Yaskawa INFORM job: R1_W27-A2(90,-90)POPR-KM-OK.JBI

/JOB
//NAME R1_W27-A2(90,-90)POPR-KM-OK
///FOLDERNAME KRIS-SCIANA
//POS
///NPOS 176,176,0,6,0,0
///TOOL 0
///POSTYPE PULSE
///PULSE
C00000=47255,92390,21974,-39561,97708,85383
C00001=10855,-90008,-88389,-33686,75537,85808
C00002=-111602,-139258,-125525,-5527,77988,-30584
C00003=-111602,-139258,-125525,-5527,77988,-30584
C00004=-63451,-99780,-87259,-34493,107645,-18593
C00005=-79235,-87779,-71168,-36428,98005,-22127
C00006=-81155,-88041,-68185,-36487,95587,-22123
C00007=-83679,-90006,-68978,-36755,94086,-22676
C00008=-83320,-89737,-68871,-36718,94298,-22597
C00009=-83320,-90271,-70181,-36754,94730,-22742
C00010=-84421,-91093,-70507,-36864,94080,-22984
C00011=-84421,-90731,-69628,-36842,93792,-22887
C00012=-81728,-89912,-71997,-36675,96467,-22659
C00013=-111602,-139258,-125525,-5527,77988,-30584
C00014=-111602,-139258,-125525,-5527,77988,-30584
C00015=-131748,-141016,-124490,10531,76516,-37016
C00016=-120565,-128207,-90021,8850,60749,-34228
C00017=-114295,-127384,-89205,7232,60054,-31882
C00018=-112834,-127008,-88848,6844,59902,-31333
C00019=-110412,-126666,-88756,6184,59829,-30410
C00020=-111525,-126835,-88802,6488,59856,-30835
C00021=-111525,-128465,-91197,6450,60489,-30798
C00022=-108910,-128023,-91079,5736,60447,-29805
C00023=-108910,-126871,-89375,5761,59994,-29827
C00024=-114109,-129808,-92766,7120,60979,-31753
C00025=-125724,-137992,-104372,9805,65099,-35816
C00026=-168598,-158328,-94882,65934,65859,5142
C00027=-138330,-90233,-84655,36621,76479,52498
C00028=-128715,-49536,-61129,33505,77884,56923
C00029=-127126,-48405,-55465,33411,74823,56634
C00030=-126813,-49148,-53910,33515,73573,56377
C00031=-126089,-49251,-53971,33315,73277,56584
C00032=-126589,-49181,-53929,33454,73482,56443
C00033=-126589,-49335,-57635,33144,75338,57009
C00034=-129344,-26255,-35376,41772,85568,55954
C00035=-129533,-29426,-35674,41853,84566,55468
C00036=-129631,-31118,-36819,41874,84489,55393
C00037=-129533,-29426,-35674,41853,84566,55468
C00038=-128070,-29028,-37630,41593,84938,56269
C00039=-124690,-38934,-42891,41199,81940,56578
C00040=-124690,-38847,-42167,41231,81636,56457
C00041=-124690,-38934,-42891,41199,81940,56578
C00042=-131035,-10866,-23942,41979,87025,55795
C00043=-124541,-12691,-28986,30832,86374,57210
C00044=-123620,-12779,-29054,30669,86041,57473
C00045=-123970,-12749,-29030,30732,86167,57373
C00046=-123970,-12682,-30414,30718,86934,57579
C00047=-120974,-15677,-32306,30215,85547,58354
C00048=-121060,-15840,-31115,30254,84866,58141
C00049=-121060,-15154,-30596,30254,84897,58150
C00050=-121060,-15840,-31115,30254,84866,58141
C00051=-121060,-15778,-32671,30227,85727,58368
C00052=-117057,-13593,-30324,29443,84053,59453
C00053=-117057,-13609,-29901,29455,83818,59392
C00054=-117057,-13593,-30324,29443,84053,59453
C00055=-124504,-18943,-37628,40859,87235,58732
C00056=-122503,-58034,-63350,23085,92729,-39111
C00057=-118561,-36204,-48728,23381,102965,-35613
C00058=-118036,-37590,-47382,23238,101399,-35730
C00059=-119514,-54944,-57534,22827,90064,-38535
C00060=-118197,-55011,-58807,22737,90395,-37994
C00061=-116993,-61076,-60812,21524,85130,-34223
C00062=-119392,-54872,-58672,22830,90711,-38368
C00063=-122456,-57021,-66004,23167,94704,-38710
C00064=-79548,-70371,-81102,-16241,84903,14397
C00065=-79548,-70265,-68951,-16505,77767,15353
C00066=-104992,-98472,-63236,13452,32992,-19166
C00067=-105182,-98024,-62675,13672,32909,-19299
C00068=-105233,-98344,-62386,13846,32587,-19397
C00069=-108042,-85190,-65154,13232,53638,-17720
C00070=-107439,-106849,-69554,15876,33022,-20670
C00071=-100440,-73805,-66430,698,65910,-23703
C00072=-75740,-68220,-64202,-17439,76767,16862
C00073=-76507,-66361,-64522,-17207,77706,16451
C00074=-94491,-76083,-67425,-3375,65969,-13243
C00075=-83535,-71278,-65200,-14735,71142,-631
C00076=-81902,-69490,-64242,-15161,71764,-113
C00077=-81635,-70718,-66741,-15162,72688,-135
C00078=-81323,-43477,-57369,-10673,89641,51992
C00079=-81466,-41816,-53340,-10647,88023,52082
C00080=-92058,-2498,-26070,-6704,90331,58112
C00081=-92407,-914,-24751,-6645,90305,57999
C00082=-92622,2167,-26871,-6629,93158,57779
C00083=-102765,8643,-22555,7262,102808,72751
C00084=-102046,12903,-14607,7435,102241,73042
C00085=-103818,11521,-15679,6623,102379,72456
C00086=-104019,13462,-16416,6672,103835,72468
C00087=-100362,7840,-23814,352,99133,73837
C00088=-93505,-42567,-98732,-7157,86742,74535
C00089=-125724,-137992,-104372,9805,65099,-35816
C00090=-110950,-137574,-92834,6542,56798,-30799
C00091=-108633,-136098,-91409,5901,56506,-29909
C00092=-110317,-120133,-87198,6027,62209,-30244
C00093=-115536,-122151,-89589,7364,63072,-32157
C00094=-115536,-142518,-126484,6818,75223,-31432
C00095=-115536,-142518,-126484,6818,75223,-31432
C00096=27632,69086,-255,32308,94480,64498
C00097=22775,131727,30764,-8837,96794,84364
C00098=23208,121491,44257,-39062,86083,83812
C00099=-45129,13731,-11238,-25738,101470,44798
C00100=-54749,18539,-6974,-25294,98453,41899
C00101=-54749,18229,-2495,-25091,95802,42470
C00102=-54749,18221,-1924,-25071,95479,42540
C00103=-54749,18229,-2495,-25091,95802,42470
C00104=-51539,33465,12284,-25169,95610,43698
C00105=-65061,29091,1530,-1828,95938,42246
C00106=-65321,28356,1709,-1805,95446,42166
C00107=-65537,27832,1195,-1788,95487,42094
C00108=-65321,28356,1709,-1805,95446,42166
C00109=-65321,28613,-146,-1811,96720,42147
C00110=-67849,26457,-1480,-1592,96380,41312
C00111=-67999,26801,118,-1576,95571,41273
C00112=-67700,25812,-843,-1602,95659,41373
C00113=-67849,26305,-364,-1589,95616,41322
C00114=-69952,33819,5307,-1407,95949,40620
C00115=-71660,37949,11429,-1253,94278,40070
C00116=-71826,38618,12117,-1238,94192,40015
C00117=-71308,36635,9188,-1286,94987,40180
C00118=-69715,46382,18396,-1423,94355,40716
C00119=-70506,44345,18212,-1352,93408,40463
C00120=-70738,43793,17625,-1334,93481,40383
C00121=-70506,44345,18212,-1352,93408,40463
C00122=-70506,44470,16366,-1355,94608,40450
C00123=-74342,36127,7664,-1021,95621,39166
C00124=-67594,51850,27286,-12922,100189,40091
C00125=-67594,51857,27602,-12911,100003,40111
C00126=-67594,51850,27286,-12922,100189,40091
C00127=-74342,37093,2887,-1031,99056,39137
C00128=-67920,8103,-14728,-23481,111043,54078
C00129=-68371,9278,-10792,-23231,109243,54283
C00130=-71989,6025,-15002,-18365,107550,55075
C00131=-68543,9839,-10380,-23257,109228,54219
C00132=-67871,11157,-7953,-23050,108659,54597
C00133=-70618,6902,-11763,-25009,100838,46496
C00134=-68309,7669,-17399,-25439,105035,46441
C00135=-36430,69905,52851,-36906,101949,40986
C00136=-36706,60275,49273,-37582,94667,38514
C00137=-36645,60382,50088,-37547,94335,38657
C00138=-37134,77452,71184,-35909,96299,43276
C00139=-36521,76032,64769,-36155,99186,42575
C00140=-48748,75637,44138,-12559,109446,36491
C00141=-47018,7632,-18403,-16315,86685,22647
C00142=-48186,9094,-11222,-16117,82930,22742
C00143=-48793,11484,-8128,-16002,82162,22634
C00144=-48845,10311,-10218,-15969,82810,22529
C00145=-48144,8977,-10156,-16147,82248,22846
C00146=-48662,11817,-7773,-16031,82142,22680
C00147=-44941,27194,6639,-21678,88433,32735
C00148=-45073,30718,10114,-21660,88092,32747
C00149=-48184,9090,-11217,-16118,82925,22743
C00150=-46490,6362,-16531,-16455,85053,23045
C00151=-51089,14800,-9249,10241,81305,-15900
C00152=-51639,15720,-5461,10436,79544,-16234
C00153=-51328,16356,-3857,10373,78855,-16186
C00154=-52394,14452,-5453,10658,78994,-16538
C00155=-51853,16186,-5099,10493,79587,-16303
C00156=-52771,20025,-2714,10728,80203,-16562
C00157=-52331,17234,-5358,10602,80335,-16402
C00158=-51787,16236,-7953,10429,81332,-16133
C00159=-102783,1332,-28831,-2508,120082,-77442
C00160=-102957,2789,-26573,-2528,119437,-77492
C00161=-101294,5159,-24044,-2166,119148,-76855
C00162=-103017,3676,-26663,-2555,119947,-77527
C00163=-103226,5472,-23865,-2576,119142,-77587
C00164=-103770,3819,-25194,-2689,119093,-77792
C00165=-103934,6110,-25506,-2765,120457,-77889
C00166=-102782,1324,-28838,-2508,120083,-77442
C00167=-102716,1959,-28722,-3690,98810,-77621
C00168=-111602,-139258,-125525,-5527,77988,-30584
C00169=-63451,-99780,-87259,-34493,107645,-18593
C00170=-77664,-93447,-72354,-35997,96893,-21092
C00171=-71109,-84007,-59579,-44165,102740,-19972
C00172=-76711,-72421,-54458,-45861,101920,-22309
C00173=-73740,-70290,-55538,-45661,104697,-22163
C00174=-73778,-73289,-89979,-52376,117942,-29543
C00175=4604,-97136,-110463,-3690,98810,-77621
BC00000=173361,170327,1069948
BC00001=285044,126360,1057855
BC00002=197925,2384,1013850
BC00003=398093,2384,1013850
BC00004=398093,2384,1013850
BC00005=398093,2384,1013850
BC00006=398093,2384,1013850
BC00007=398093,2384,1013850
BC00008=398093,2384,1013850
BC00009=398093,2384,1013850
BC00010=398093,2384,1013850
BC00011=398093,2384,1013850
BC00012=398093,2384,1013850
BC00013=398093,2384,1013850
BC00014=197925,2384,1013850
BC00015=16093,2384,1007970
BC00016=16093,2384,1007970
BC00017=16093,2384,1007970
BC00018=16093,2384,1007970
BC00019=16093,2384,1007970
BC00020=16093,2384,1007970
BC00021=16093,2384,1007970
BC00022=16093,2384,1007970
BC00023=16093,2384,1007970
BC00024=16093,2384,1007970
BC00025=16093,2384,1007970
BC00026=2663,3711,1022453
BC00027=269,7512,1047096
BC00028=269,7512,1047096
BC00029=269,7512,1047096
BC00030=269,7512,1047096
BC00031=269,7512,1047096
BC00032=269,7512,1047096
BC00033=269,7512,1047096
BC00034=15,11820,1075020
BC00035=15,11820,1075020
BC00036=15,11820,1075020
BC00037=15,11820,1075020
BC00038=15,11820,1075020
BC00039=15,11820,1075020
BC00040=15,11820,1075020
BC00041=15,11820,1075020
BC00042=15,11820,1075020
BC00043=15,11820,1075020
BC00044=15,11820,1075020
BC00045=15,11820,1075020
BC00046=15,11820,1075020
BC00047=15,11820,1075020
BC00048=15,11820,1075020
BC00049=15,11820,1075020
BC00050=15,11820,1075020
BC00051=15,11820,1075020
BC00052=15,11820,1075020
BC00053=15,11820,1075020
BC00054=15,11820,1075020
BC00055=15,11820,1075020
BC00056=15,49099,1075175
BC00057=15,47349,1075175
BC00058=15,47349,1075175
BC00059=15,47349,1075175
BC00060=15,47349,1075175
BC00061=15,62077,1075175
BC00062=15,62577,1075175
BC00063=15,63827,1075175
BC00064=15,12213,1075175
BC00065=15,12213,1075175
BC00066=16,12213,1075171
BC00067=16,12213,1075171
BC00068=16,12213,1075171
BC00069=16,12213,1075171
BC00070=16,12213,1075171
BC00071=16,12213,1075171
BC00072=15,16755,1075175
BC00073=15,16755,1075175
BC00074=16,12213,1075171
BC00075=16,12213,1075171
BC00076=16,12213,1075171
BC00077=16,12213,1075171
BC00078=16,12213,1075171
BC00079=16,12213,1075171
BC00080=16,12213,1075171
BC00081=16,12213,1075171
BC00082=16,12213,1075171
BC00083=17,22433,1075169
BC00084=17,22433,1075167
BC00085=17,22433,1075169
BC00086=17,22433,1075169
BC00087=16,12213,1075171
BC00088=16,12213,1075171
BC00089=16093,2384,1007970
BC00090=16093,2384,1007970
BC00091=16093,2384,1007970
BC00092=16093,2384,1007970
BC00093=16093,2384,1007970
BC00094=16093,2384,1007970
BC00095=92875,102,1007970
BC00096=25030,15919,1060143
BC00097=103306,16446,1075157
BC00098=79646,13110,1075161
BC00099=246913,5043,1075175
BC00100=246913,5043,1075175
BC00101=246913,5043,1075175
BC00102=246913,5043,1075175
BC00103=246913,5043,1075175
BC00104=246913,5043,1075175
BC00105=246913,5043,1075175
BC00106=246913,5043,1075175
BC00107=246913,5043,1075175
BC00108=246913,5043,1075175
BC00109=246913,5043,1075175
BC00110=246913,5043,1075175
BC00111=246913,5043,1075175
BC00112=246913,5043,1075175
BC00113=246913,5043,1075175
BC00114=246913,5043,1075175
BC00115=246913,5043,1075175
BC00116=246913,5043,1075175
BC00117=246913,5043,1075175
BC00118=246913,5043,1075175
BC00119=246913,5043,1075175
BC00120=246913,5043,1075175
BC00121=246913,5043,1075175
BC00122=246913,5043,1075175
BC00123=246913,5043,1075175
BC00124=246913,5043,1075175
BC00125=246913,5043,1075175
BC00126=246913,5043,1075175
BC00127=246913,5043,1075175
BC00128=310215,25331,1075175
BC00129=304559,24148,1075175
BC00130=304559,24148,1075175
BC00131=302296,23674,1075175
BC00132=302296,23674,1075175
BC00133=304559,24148,1075175
BC00134=304559,24148,1075175
BC00135=197323,15,1075175
BC00136=197323,15,1075175
BC00137=197323,15,1075175
BC00138=197323,15,1075175
BC00139=197323,15,1075175
BC00140=197323,15,1075175
BC00141=197986,15,1075175
BC00142=197986,15,1075175
BC00143=197986,15,1075175
BC00144=198252,15,1075175
BC00145=198252,15,1075175
BC00146=200364,15,1075175
BC00147=200364,15,1075175
BC00148=200364,15,1075175
BC00149=200098,15,1075175
BC00150=199434,15,1075175
BC00151=148787,33401,1075175
BC00152=154351,32151,1075175
BC00153=156150,31747,1075172
BC00154=156576,31651,1075175
BC00155=156576,31651,1075175
BC00156=156716,69750,1059420
BC00157=154490,70250,1066913
BC00158=148927,71500,1075175
BC00159=344706,64580,1052547
BC00160=343940,58320,1037184
BC00161=343634,55816,1031039
BC00162=343634,55816,1031039
BC00163=343634,55816,1031039
BC00164=343634,55816,1031039
BC00165=343634,55816,1031039
BC00166=341638,64598,1052619
BC00167=341637,64597,1052617
BC00168=398093,160168,1013850
BC00169=398093,2384,1013850
BC00170=398093,2384,1013850
BC00171=398093,2384,1013850
BC00172=398093,2384,1013850
BC00173=398093,2384,1013850
BC00174=398093,2384,1013850
BC00175=176985,505314,1052617
///POSTYPE BASE
///RECTAN
///RCONF 0,0,0,0,1,0,0,0,0,0,0,0,0,0,0,0,0,0,0,0,0,0,0,0
P00006=2.006,1.622,-0.565,0.0000,0.0000,0.0000
///RCONF 0,0,0,0,0,0,0,0,0,0,0,0,0,0,0,0,0,0,0,0,0,0,0,0
P00023=-2.957,-4.083,2.762,0.0000,0.0000,0.0000
P00024=-1.466,-0.226,-0.419,0.0000,0.0000,0.0000
P00025=3.643,0.007,-2.585,0.0000,0.0000,0.0000
P00040=2.716,-0.016,3.014,0.0000,0.0000,0.0000
P00041=-0.109,0.014,0.966,0.0000,0.0000,0.0000
//INST
///DATE 2025/02/21 10:28
///ATTR SC,RW
///GROUP1 RB1,BS1
NOP
SFTOF
MOVJ C00000 BC00000 VJ=100.00
MOVJ C00001 BC00001 VJ=100.00
MOVJ C00002 BC00002 VJ=100.00
'DODANO BP 060624
MOVJ C00003 BC00003 VJ=100.00
MOVJ C00004 BC00004 VJ=100.00
MOVL C00005 BC00005 V=233.3
MOVL C00006 BC00006 V=60.0
REFP 3 C00007 BC00007
CALL JOB:SEARCH-R1
SET P040 P006
SFTON P040
MOVL C00008 BC00008 V=100.0
MOVL C00009 BC00009 V=100.0
MOVL C00010 BC00010 V=60.0
REFP 3 C00011 BC00011
CALL JOB:SEARCH-R1
SET P040 P006
SFTON P040
MOVL C00012 BC00012 V=100.0
MOVJ C00013 BC00013 VJ=100.00
MOVJ C00014 BC00014 VJ=100.00
MOVL C00015 BC00015 V=666.7
MOVL C00016 BC00016 V=666.7
MOVL C00017 BC00017 V=233.3
MOVL C00018 BC00018 V=60.0
REFP 3 C00019 BC00019
CALL JOB:SEARCH-R1
SET P041 P006
SFTON P041
MOVL C00020 BC00020 V=100.0
MOVL C00021 BC00021 V=100.0
MOVL C00022 BC00022 V=60.0
REFP 3 C00023 BC00023
CALL JOB:SEARCH-R1
SET P041 P006
SFTON P041
MOVL C00024 BC00024 V=100.0
MOVL C00025 BC00025 V=666.7
'KONIEC BP 060624
MOVJ C00026 BC00026 VJ=100.00
MOVJ C00027 BC00027 VJ=100.00
MOVJ C00028 BC00028 VJ=100.00
MOVJ C00029 BC00029 VJ=100.00
MOVL C00030 BC00030 V=60.0
REFP 3 C00031 BC00031
CALL JOB:SEARCH-R1
SET P023 P006
SFTON P023
MOVL C00032 BC00032 V=60.0
MOVL C00033 BC00033 V=100.0
MOVL C00034 BC00034 V=100.0
MOVL C00035 BC00035 V=100.0
REFP 3 C00036 BC00036
CALL JOB:SEARCH-R1
SET P023 P006
SFTON P023
MOVL C00037 BC00037 V=60.0
MOVL C00038 BC00038 V=100.0
MOVL C00039 BC00039 V=100.0
REFP 3 C00040 BC00040
CALL JOB:SEARCH-R1
SET P023 P006
SFTON P023
MOVL C00041 BC00041 V=60.0
'DRUGI NOWY POMIAR
SFTOF
MOVL C00042 BC00042 V=100.0
MOVL C00043 BC00043 V=100.0
REFP 3 C00044 BC00044
CALL JOB:SEARCH-R1
SET P024 P006
SFTON P024
MOVL C00045 BC00045 V=60.0
MOVL C00046 BC00046 V=100.0
MOVL C00047 BC00047 V=100.0
MOVL C00048 BC00048 V=60.0
REFP 3 C00049 BC00049
CALL JOB:SEARCH-R1
SET P024 P006
SFTON P024
MOVL C00050 BC00050 V=60.0
MOVL C00051 BC00051 V=100.0
MOVL C00052 BC00052 V=60.0
REFP 3 C00053 BC00053
CALL JOB:SEARCH-R1
SET P024 P006
SFTON P024
MOVL C00054 BC00054 V=60.0
MOVJ C00055 BC00055 VJ=30.00
SFTOF
'Path W988
SFTOF
SFTON P023
CALL JOB:COFNIJ_DRUT
MOVJ C00056 BC00056 VJ=50.00
MOVJ C00057 BC00057 VJ=100.00
MOVL C00058 BC00058 V=100.0 PL=0
REFP 1 C00059 BC00059
REFP 2 C00060 BC00060
MACRO1 MJ#(0) ARGF7
ARCON
SFTON P024
MOVL C00061 BC00061 V=10.8
ARCOF
MOVL C00062 BC00062 V=100.0
MOVJ C00063 BC00063 VJ=50.00
SFTOF
'Path W989
SFTOF
SFTON P023
MOVJ C00064 BC00064 VJ=100.00
MOVJ C00065 BC00065 VJ=50.00
MOVL C00066 BC00066 V=100.0
ARCON
MOVL C00067 BC00067 V=8.3
MOVL C00068 BC00068 V=8.3
MOVL C00069 BC00069 V=8.3
ARCOF
SFTOF
MOVL C00070 BC00070 V=83.3
SFTON P023
MOVL C00071 BC00071 V=100.0 PL=0
REFP 1 C00072 BC00072
REFP 2 C00073 BC00073
MACRO1 MJ#(0) ARGF7
ARCON
TIMER T=0.50
MOVL C00074 BC00074 V=10.0
MOVL C00075 BC00075 V=10.0
MOVL C00076 BC00076 V=10.0
ARCOF
MOVJ C00077 BC00077 VJ=15.00
MOVJ C00078 BC00078 VJ=100.00
MOVJ C00079 BC00079 VJ=100.00
ARCON
SFTON P024
MOVL C00080 BC00080 V=10.0
MOVL C00081 BC00081 V=10.0
ARCOF
MOVJ C00082 BC00082 VJ=15.00
MOVJ C00083 BC00083 VJ=100.00
MOVJ C00084 BC00084 VJ=20.00
ARCON
MOVL C00085 BC00085 V=10.0
ARCOF
MOVL C00086 BC00086 V=100.0
MOVL C00087 BC00087 V=166.7
MOVJ C00088 BC00088 VJ=100.00
SFTOF
'BP 060624
MOVJ C00089 BC00089 VJ=100.00
MOVJ C00090 BC00090 VJ=100.00
SFTON P041
MOVL C00091 BC00091 V=100.0 PL=0
MACRO1 MJ#(0) ARGF6
ARCON
MOVL C00092 BC00092 V=11.7
ARCOF
MOVL C00093 BC00093 V=11.7
SFTOF
MOVL C00094 BC00094 V=666.7
MOVL C00095 BC00095 V=666.7
'KONIEC BP 060624
'2 STRONA
MOVJ C00096 BC00096 VJ=100.00
'Path VIA1124
SFTOF
MOVJ C00097 BC00097 VJ=100.00
CALL JOB:ONLYCUT-R1_LONG
'Path S992
SFTOF
MOVJ C00098 BC00098 VJ=100.00
SFTOF
MOVJ C00099 BC00099 VJ=100.00
MOVJ C00100 BC00100 VJ=100.00
MOVL C00101 BC00101 V=83.3
REFP 3 C00102 BC00102
CALL JOB:SEARCH-R1
SET P024 P006
SFTON P024
MOVL C00103 BC00103 V=60.0
MOVL C00104 BC00104 V=100.0
MOVL C00105 BC00105 V=100.0
MOVL C00106 BC00106 V=100.0
REFP 3 C00107 BC00107
CALL JOB:SEARCH-R1
SET P024 P006
SFTON P024
MOVL C00108 BC00108 V=60.0
MOVL C00109 BC00109 V=100.0
MOVL C00110 BC00110 V=83.3
MOVL C00111 BC00111 V=100.0
REFP 3 C00112 BC00112
CALL JOB:SEARCH-R1
SET P024 P006
SFTON P024
MOVL C00113 BC00113 V=60.0
SFTOF
MOVL C00114 BC00114 V=100.0
MOVL C00115 BC00115 V=100.0
REFP 3 C00116 BC00116
CALL JOB:SEARCH-R1
SET P025 P006
SFTON P025
MOVL C00117 BC00117 V=100.0
MOVL C00118 BC00118 V=100.0
MOVL C00119 BC00119 V=100.0
REFP 3 C00120 BC00120
CALL JOB:SEARCH-R1
SET P025 P006
SFTON P025
MOVL C00121 BC00121 V=100.0
MOVL C00122 BC00122 V=100.0
MOVL C00123 BC00123 V=100.0
MOVL C00124 BC00124 V=100.0
REFP 3 C00125 BC00125
CALL JOB:SEARCH-R1
SET P025 P006
SFTON P025
MOVL C00126 BC00126 V=100.0
MOVL C00127 BC00127 V=100.0
'Path W993
SFTOF
SFTON P024
MOVJ C00128 BC00128 VJ=100.00
MOVJ C00129 BC00129 VJ=100.00
SFTON P024
MOVL C00130 BC00130 V=100.0 PL=0
REFP 1 C00131 BC00131
REFP 2 C00132 BC00132
MACRO1 MJ#(0) ARGF7
ARCON
SFTON P025
MOVL C00133 BC00133 V=10.0
ARCOF
MOVL C00134 BC00134 V=100.0
SFTOF
SFTON P024
MOVJ C00135 BC00135 VJ=20.00
MOVJ C00136 BC00136 VJ=20.00
ARCON
MOVL C00137 BC00137 V=8.3
MOVL C00138 BC00138 V=8.3
ARCOF
MOVL C00139 BC00139 V=83.3
MOVJ C00140 BC00140 VJ=20.00
MOVJ C00141 BC00141 VJ=20.00
MOVJ C00142 BC00142 VJ=100.00
SFTON P024
MOVL C00143 BC00143 V=100.0 PL=0
REFP 1 C00144 BC00144
REFP 2 C00145 BC00145
MACRO1 MJ#(0) ARGF7
ARCON
MOVL C00146 BC00146 V=10.0
MOVL C00147 BC00147 V=10.0
MOVL C00148 BC00148 V=10.0
ARCOF
MOVL C00149 BC00149 V=100.0
MOVL C00150 BC00150 V=166.7
SFTOF
'Path W995
SFTOF
SFTON P024
MOVJ C00151 BC00151 VJ=100.00
MOVJ C00152 BC00152 VJ=100.00
SFTON P024
MOVL C00153 BC00153 V=100.0 PL=0
REFP 1 C00154 BC00154
REFP 2 C00155 BC00155
MACRO1 MJ#(0) ARGF7
ARCON
SFTON P025
MOVL C00156 BC00156 V=10.0
ARCOF
MOVL C00157 BC00157 V=400.0
MOVL C00158 BC00158 V=1000.0
SFTOF
MOVJ C00159 BC00159 VJ=100.00
MOVJ C00160 BC00160 VJ=100.00
SFTON P025
MOVL C00161 BC00161 V=100.0 PL=0
REFP 1 C00162 BC00162
REFP 2 C00163 BC00163
MACRO1 MJ#(0) ARGF7
ARCON
MOVL C00164 BC00164 V=10.0
ARCOF
MOVL C00165 BC00165 V=100.0
MOVL C00166 BC00166 V=166.7
SFTOF
MOVJ C00167 BC00167 VJ=100.00
'BP 060624
SFTOF
MOVL C00168 BC00168 V=666.7
MOVL C00169 BC00169 V=666.7
MOVL C00170 BC00170 V=666.7
SFTON P040
MOVL C00171 BC00171 V=100.0 PL=0
MACRO1 MJ#(0) ARGF6
ARCON
MOVL C00172 BC00172 V=11.7
ARCOF
MOVL C00173 BC00173 V=266.7
SFTOF
MOVJ C00174 BC00174 VJ=100.00
'KONIEC BP 060624
MOVJ C00175 BC00175 VJ=100.00
END
